Universal Robots PolyScope program: a_to_g.urp

Program a_to_g (installation=string_planes directory=/programs/string_crossings createdIn=5.17.3 lastSavedIn=5.17.3 robotSerialNumber=20245501435)
Calibrated DH parameters: a=[0.000154, -0.137004, -0.385524, -0.00002, 0.000092, 0]; d=[0.162441, 211.794786, -230.585024, 18.923638, 0.099786, 0.09951]; alpha=[1.569493, -0.001902, 0.003874, 1.570111, -1.570167, 0]; deltaTheta=[0, -1.242934, 1.056292, 0.186646, 0.000002, 0.000001]
InitVariablesNode
Robot Program (runOnlyOnce=false)
  bow_section := -1
  If bow_section≟-1
    MoveJ speed 60 deg/s, acceleration 80 deg/s^2 (useActiveTCP=true) feature=Base
      Waypoint Waypoint_2 (Relative): relativeFromPosition TCP in base x=277.254 y=734.024 z=156.891 mm, rx=1.739 ry=2.3104 rz=-1.1077 rad; joints [-126.649, -28.124, 54.73, -74.617, -91.964, -141.812] deg; TCP offset x=28.21 y=-96.107 z=-99.69 mm, rx=0 ry=0 rz=0 rad; TCP in base x=333.304 y=655.498 z=103.667 mm, rx=-1.6491 ry=-1.7982 rz=0.6657 rad; joints [-132.463, -27.758, 71.844, -100.482, -56.045, -147.728] deg
  ElseIf bow_section≟0
    MoveJ speed 60 deg/s, acceleration 80 deg/s^2 (useActiveTCP=true) feature=Base
      Waypoint Waypoint_1 (Relative): relativeFromPosition TCP in base x=327.375 y=541.709 z=231.859 mm, rx=1.6817 ry=2.3248 rz=-1.1115 rad; joints [-139.64, -50.32, 85.997, -84.694, -102.36, -153.081] deg; TCP in base x=267.746 y=455.84 z=63.354 mm, rx=-1.6064 ry=-1.9108 rz=0.8701 rad; joints [-141.612, -39.193, 108.911, -115.29, -70.78, -159.12] deg
  Else 
    MoveJ speed 60 deg/s, acceleration 80 deg/s^2 (useActiveTCP=true) feature=Base
      Waypoint Waypoint_3 (Relative): relativeFromPosition TCP in base x=374.965 y=359.139 z=303.04 mm, rx=1.6275 ry=2.3374 rz=-1.1145 rad; joints [-156.115, -66.368, 101.551, -88.734, -114.428, -168.118] deg; TCP in base x=243.614 y=214.06 z=64.414 mm, rx=-1.5873 ry=-1.9212 rz=0.9621 rad; joints [-169.308, -44.603, 138.126, -133.881, -94.42, -177.776] deg
